# EPICS substitutions: ioc-repository/test/startup/db/test.substitutions
file db/ramper.db {
    pattern { name }
        { xxx }
}
